FUNCTION_BLOCK FB_RecipeBuilderBorgoFlaps EXTENDS FB_RecipeBase

METHOD Build : BOOL
VAR_INST
    TotalY          : REAL;
    TotalX          : REAL;
    ShorterY        : REAL;
    ShorterX        : REAL;
END_VAR
// ==========================================================
//  Recepta testowa
// ==========================================================

TotalY   := _Config.PanelFrontLength + 2 * _Config.PanelHeight;
TotalX   := _Config.PanelFrontWidth  + 2 * _Config.PanelHeight; 
ShorterY := TotalY - _Config.PanelHeight;
ShorterX := TotalX - _Config.PanelHeight;
_FootprintX := TotalX;
_FootprintY := TotalY;
_MaxCopiesX := DINT_TO_INT(TRUNC(RAW_BOARD_X / _FootprintX));
_MaxCopiesY := DINT_TO_INT(TRUNC(RAW_BOARD_Y / _FootprintY));

IF _Config.FillAll THEN
    _ActualCopiesX := _MaxCopiesX;
    _ActualCopiesY := _MaxCopiesY;
ELSE
    // Jeśli nie "wypełnij", to bierzemy to co chce operator, ale obcinamy od 1 do Max!
    _ActualCopiesX := LIMIT(1, _Config.RequestedCopiesX, _MaxCopiesX);
    _ActualCopiesY := LIMIT(1, _Config.RequestedCopiesY, _MaxCopiesY);
END_IF

_SegmentsToGroove := 0;

_SegmentsToCutX   := 2;

_SegmentsCutX[1].Start.X := TotalX;
_SegmentsCutX[1].Stop.X  := 0;
_SegmentsCutX[1].Start.Y := TotalY;
_SegmentsCutX[1].Stop.Y  := TotalY;

_SegmentsCutX[2].Start.X := TotalX;
_SegmentsCutX[2].Stop.X  := 0;
_SegmentsCutX[2].Start.Y := 0;
_SegmentsCutX[2].Stop.Y  := 0;

_SegmentsToCutY   := 2;

_SegmentsCutY[1].Start.X := TotalX;
_SegmentsCutY[1].Stop.X  := TotalX;
_SegmentsCutY[1].Start.Y := TotalY;
_SegmentsCutY[1].Stop.Y  := 0;

_SegmentsCutY[2].Start.X := 0;
_SegmentsCutY[2].Stop.X  := 0;
_SegmentsCutY[2].Start.Y := TotalY;
_SegmentsCutY[2].Stop.Y  := 0;



Build := TRUE;
END_METHOD

METHOD FB_init : BOOL
VAR_INPUT
	bInitRetains : BOOL; // if TRUE, the retain variables are initialized (warm start / cold start)
	bInCopyCode : BOOL;  // if TRUE, the instance afterwards gets moved into the copy code (online change)
END_VAR
_Limits.PanelFrontLength.MinVal := 12.0;
_Limits.PanelFrontLength.MaxVal := 1234.0;

_Limits.PanelFrontWidth.MinVal  := 12.0;
_Limits.PanelFrontWidth.MaxVal  := 1234.0;

_Limits.PanelHeight.MinVal      := 12.0;
_Limits.PanelHeight.MaxVal      := 1234.0;

_Limits.RailHeightCorrection.MinVal := 12.0;
_Limits.RailHeightCorrection.MaxVal := 1234.0;

_Limits.CuttingOverpass.MinVal := 0.0;
_Limits.CuttingOverpass.MaxVal := 50.0;

_Limits.GroovingOverpass.MinVal := 0.0;
_Limits.GroovingOverpass.MaxVal := 50.0;
END_METHOD

METHOD UpdateNestingLimits
VAR
    TotalX : REAL;
    TotalY : REAL;
END_VAR


// Liczymy Footprint "w locie"
TotalX := _Config.PanelFrontWidth  + 2 * _Config.PanelHeight; 
TotalY := _Config.PanelFrontLength + 2 * _Config.PanelHeight;

_FootprintX := TotalX;
_FootprintY := TotalY;

IF _FootprintX > 0.0 THEN
    _MaxCopiesX := REAL_TO_DINT(TRUNC(RAW_BOARD_X / _FootprintX));
ELSE
    _MaxCopiesX := 1;
END_IF

IF _FootprintY > 0.0 THEN
    _MaxCopiesY := REAL_TO_DINT(TRUNC(RAW_BOARD_Y / _FootprintY));
ELSE
    _MaxCopiesY := 1;
END_IF

// Zabezpieczenie przed bzdurami
IF _MaxCopiesX < 1 THEN _MaxCopiesX := 1; END_IF
IF _MaxCopiesY < 1 THEN _MaxCopiesY := 1; END_IF

// Update limitów dla wizualizacji (Numpad HMI)
_Limits.RequestedCopiesX.MinVal := 1.0;
_Limits.RequestedCopiesX.MaxVal := DINT_TO_REAL(_MaxCopiesX);

_Limits.RequestedCopiesY.MinVal := 1.0;
_Limits.RequestedCopiesY.MaxVal := DINT_TO_REAL(_MaxCopiesY);
END_METHOD

END_FUNCTION_BLOCK

(* stored: Version 1.1.0.1, ProductVersion 3.1.4024.15
   POU FB_RecipeBuilderBorgoFlaps: Id {1389b747-8c88-4122-8f76-112cbf46c424}, SpecialFunc None
   Method Build: Id {a7636aac-6540-4877-9111-d7366342a8fe}
   Method FB_init: Id {4a0331ae-cce1-43c4-8f3f-519ce38c4c04}
   Method UpdateNestingLimits: Id {2b71f6ce-b964-482a-9b7f-2de722577ce3} *)
